INTERFACE I_ChunkedResponseManagerConfig

METHOD PUBLIC TryGetResponseIdFromRequest : BOOL
VAR_INPUT
	Request : I_Request;
	Destination : ANY;
END_VAR
END_METHOD

METHOD PUBLIC TryGetSessionIdFromRequest : BOOL
VAR_INPUT
	Request : I_Request;
	Destination : ANY;
END_VAR
END_METHOD

METHOD PUBLIC TryGetSessionIdFromResponse : BOOL
VAR_INPUT
	Response : I_ServerResponse;
	Destination : ANY;
END_VAR
END_METHOD

METHOD PUBLIC UpdateResponseWithHasMoreChunks
VAR_INPUT
	Response : I_ServerResponse;
	ResponseId : T_MAXSTRING;
END_VAR
END_METHOD

END_INTERFACE

(* stored: Version 1.1.0.1, ProductVersion 3.1.4024.12
   Itf I_ChunkedResponseManagerConfig: Id {2ab1b2b2-5d42-4352-9af9-83e67d269662}
   Method TryGetResponseIdFromRequest: Id {d5c64733-9d8b-4aee-b144-ef905db36ad0}
   Method TryGetSessionIdFromRequest: Id {0d7a3b18-d6b5-47d7-8281-4210b63e9db0}
   Method TryGetSessionIdFromResponse: Id {8240d26d-1ee8-4b53-869c-0f2d202f5dfe}
   Method UpdateResponseWithHasMoreChunks: Id {3ff718b8-82be-4a55-a9cf-84a074eafbc7} *)
